// TIA Portal V21 export
// export: Created 2026-07-05T03:49:26.3917626Z, ExportSetting None, DisplayName Totally Integrated Automation Portal, DisplayVersion V21, DisplayName SINAMICS Startdrive Advanced, DisplayVersion V21, DisplayName SINAMICS Startdrive G110M, G120, G120C, G120D, G120P, G115D, DisplayVersion V21, DisplayName SINAMICS Startdrive G130, G150, S120, S150, G200, G220, S200, S210, S220, Innomotics MVD, DisplayVersion V21, DisplayName STEP 7 Professional, DisplayVersion V21, DisplayName STEP 7 Safety, DisplayVersion V21, DisplayName Tech WebApplication, DisplayVersion V21, DisplayName WinCC Basic/Comfort/Advanced, DisplayVersion V21, DisplayName WinCC Professional, DisplayVersion V21, DisplayName WinCC Unified, DisplayVersion V21
FUNCTION_BLOCK "FlowControl_LAD"   // FB2100, LAD
{ S7_Optimized_Access := 'TRUE' }
// stored: AutoNumber false, MemoryReserve 100, SetENOAutomatically false
   VAR_INPUT
      启用 : Bool;   // 使能流程控制FB，FALSE时不允许启动
      启动 : Bool;   // 启动命令，条件满足时进入步骤1
      停止 : Bool;   // 正常停止命令，停止运行并把当前步清零
      暂停 : Bool;   // 暂停命令，保持当前步不继续推进
      复位 : Bool;   // 复位命令，清除完成/故障/暂停并把当前步清零
      中止 : Bool;   // 中止命令，强制退出流程并把当前步清零
      启动允许 : Bool;   // 启动允许条件，例如安全、气压、伺服Ready等
      联锁正常 : Bool;   // 运行中联锁正常，FALSE时触发故障
   END_VAR
   VAR_OUTPUT
      就绪 : Bool;   // 可启动状态：启用、允许、无运行、无故障、未完成
      运行中 : Bool;   // 流程运行锁存状态
      完成 : Bool;   // 流程正常完成，需要复位清除
      故障 : Bool;   // 流程异常停止，需要复位清除
      已暂停 : Bool;   // 流程暂停锁存状态
      当前步 : Int;   // 当前流程步骤号，流程段直接MOVE维护
      故障代码 : Word;   // 故障代码，257表示运行中联锁断开
   END_VAR
   VAR
      启动边沿 : Bool;   // 启动P上升沿指令的边沿存储位
      完成边沿 : Bool;   // 完成P上升沿线圈的边沿存储位
      执行条件 : Bool;   // 运行中和未暂停映射给执行条件
      IEC_Timer_0_Instance { S7_SetPoint := 'True'} : TON_TIME;
      IEC_Timer_0_Instance_1 { S7_SetPoint := 'True'} : TON_TIME;
   END_VAR
   VAR_TEMP   // added for the SCL form of the ladder/FBD networks
      _w1 : Bool;
      _w2 : Bool;
   END_VAR
BEGIN

REGION Network 1: 复位或中止清除流程状态
   // 复位或中止时一次性清除运行、暂停、完成、故障、当前步和故障代码。
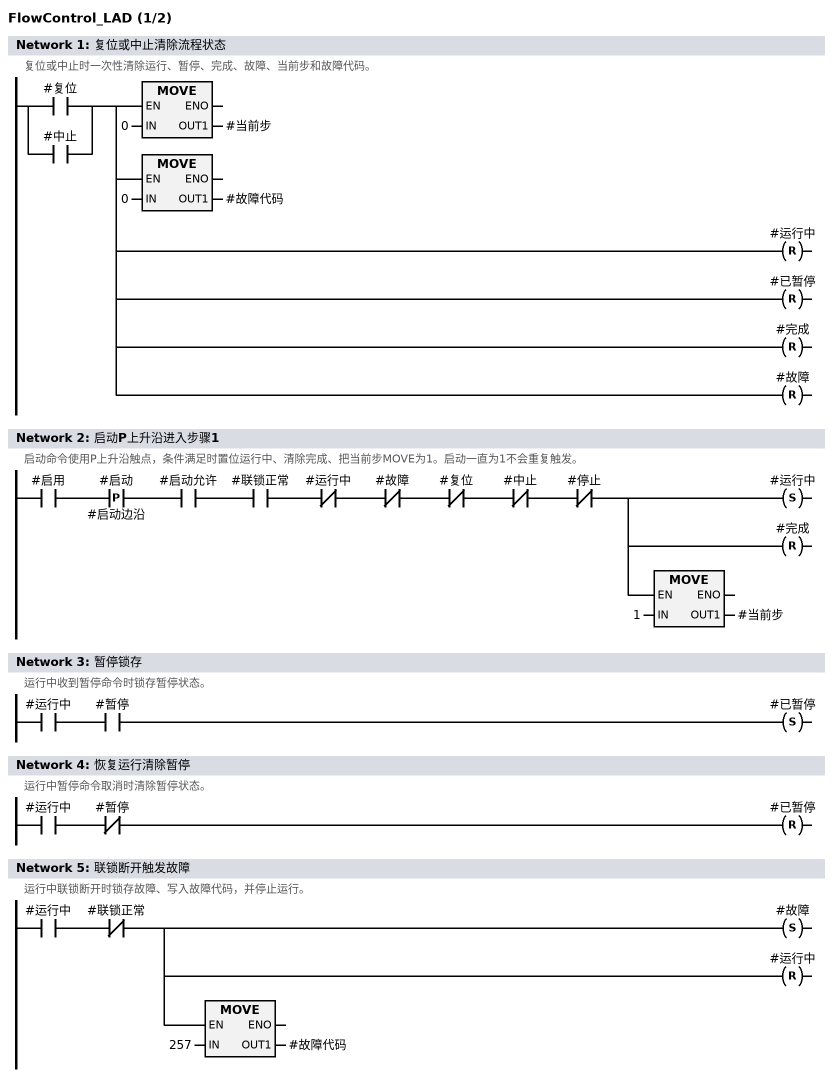
   RUNG wire#powerrail
      Contact( #复位 )
      wire#w1
      { S7_GenerateENO := "TRUE" } Move(in := 0, out1 => #当前步)
   END_RUNG
   RUNG wire#powerrail
      Contact( #中止 )
   END_RUNG wire#w1
   RUNG wire#w1
      { S7_GenerateENO := "TRUE" } Move(in := 0, out1 => #故障代码)
   END_RUNG
   RUNG wire#w1
      R_Coil( #运行中 )
   END_RUNG
   RUNG wire#w1
      R_Coil( #已暂停 )
   END_RUNG
   RUNG wire#w1
      R_Coil( #完成 )
   END_RUNG
   RUNG wire#w1
      R_Coil( #故障 )
   END_RUNG
   // the same network as SCL:
   IF #复位 OR #中止 THEN
       #当前步 := 0;
       #故障代码 := 0;
       #运行中 := FALSE;
       #已暂停 := FALSE;
       #完成 := FALSE;
       #故障 := FALSE;
   END_IF;
END_REGION

REGION Network 2: 启动P上升沿进入步骤1
   // 启动命令使用P上升沿触点，条件满足时置位运行中、清除完成、把当前步MOVE为1。启动一直为1不会重复触发。
   RUNG wire#powerrail
      Contact( #启用 )
      P_Contact(operand := #启动, bit := #启动边沿)
      Contact( #启动允许 )
      Contact( #联锁正常 )
      I_Contact( #运行中 )
      I_Contact( #故障 )
      I_Contact( #复位 )
      I_Contact( #中止 )
      I_Contact( #停止 )
      wire#w1
      S_Coil( #运行中 )
   END_RUNG
   RUNG wire#w1
      R_Coil( #完成 )
   END_RUNG
   RUNG wire#w1
      { S7_GenerateENO := "TRUE" } Move(in := 1, out1 => #当前步)
   END_RUNG
   // the same network as SCL:
   #_w1 := #启用 AND #启动 AND NOT #启动边沿;   // rising edge of #启动
   #启动边沿 := #启动;
   #_w2 := #_w1 AND #启动允许 AND #联锁正常 AND NOT #运行中 AND NOT #故障 AND NOT #复位 AND NOT #中止 AND NOT #停止;
   IF #_w2 THEN
       #运行中 := TRUE;
       #完成 := FALSE;
       #当前步 := 1;
   END_IF;
END_REGION

REGION Network 3: 暂停锁存
   // 运行中收到暂停命令时锁存暂停状态。
   RUNG wire#powerrail
      Contact( #运行中 )
      Contact( #暂停 )
      S_Coil( #已暂停 )
   END_RUNG
   // the same network as SCL:
   IF #运行中 AND #暂停 THEN #已暂停 := TRUE; END_IF;
END_REGION

REGION Network 4: 恢复运行清除暂停
   // 运行中暂停命令取消时清除暂停状态。
   RUNG wire#powerrail
      Contact( #运行中 )
      I_Contact( #暂停 )
      R_Coil( #已暂停 )
   END_RUNG
   // the same network as SCL:
   IF #运行中 AND NOT #暂停 THEN #已暂停 := FALSE; END_IF;
END_REGION

REGION Network 5: 联锁断开触发故障
   // 运行中联锁断开时锁存故障、写入故障代码，并停止运行。
   RUNG wire#powerrail
      Contact( #运行中 )
      I_Contact( #联锁正常 )
      wire#w1
      S_Coil( #故障 )
   END_RUNG
   RUNG wire#w1
      R_Coil( #运行中 )
   END_RUNG
   RUNG wire#w1
      { S7_GenerateENO := "TRUE" } Move(in := 257, out1 => #故障代码)
   END_RUNG
   // the same network as SCL:
   IF #运行中 AND NOT #联锁正常 THEN #故障 := TRUE; END_IF;
   #_w1 := #运行中 AND NOT #联锁正常;
   IF #_w1 THEN
       #运行中 := FALSE;
       #故障代码 := 257;
   END_IF;
END_REGION

REGION Network 6: 停止命令停止流程
   // 停止命令复位运行中，并把当前步MOVE为0。
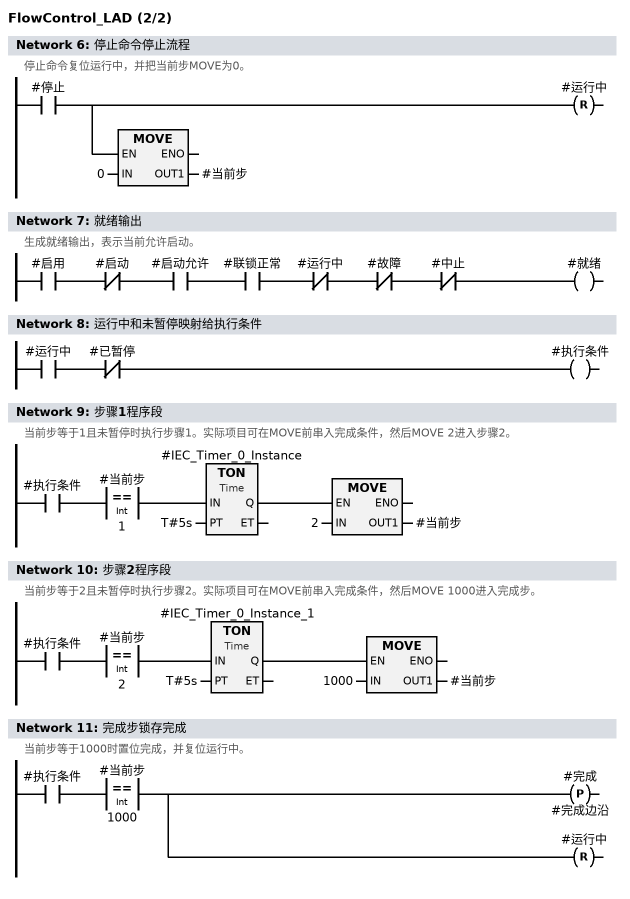
   RUNG wire#powerrail
      Contact( #停止 )
      wire#w1
      R_Coil( #运行中 )
   END_RUNG
   RUNG wire#w1
      { S7_GenerateENO := "TRUE" } Move(in := 0, out1 => #当前步)
   END_RUNG
   // the same network as SCL:
   IF #停止 THEN
       #运行中 := FALSE;
       #当前步 := 0;
   END_IF;
END_REGION

REGION Network 7: 就绪输出
   // 生成就绪输出，表示当前允许启动。
   RUNG wire#powerrail
      Contact( #启用 )
      I_Contact( #启动 )
      Contact( #启动允许 )
      Contact( #联锁正常 )
      I_Contact( #运行中 )
      I_Contact( #故障 )
      I_Contact( #中止 )
      Coil( #就绪 )
   END_RUNG
   // the same network as SCL:
   #就绪 := #启用 AND NOT #启动 AND #启动允许 AND #联锁正常 AND NOT #运行中 AND NOT #故障 AND NOT #中止;
END_REGION

REGION Network 8: 运行中和未暂停映射给执行条件
   RUNG wire#powerrail
      Contact( #运行中 )
      I_Contact( #已暂停 )
      Coil( #执行条件 )
   END_RUNG
   // the same network as SCL:
   #执行条件 := #运行中 AND NOT #已暂停;
END_REGION

REGION Network 9: 步骤1程序段
   // 当前步等于1且未暂停时执行步骤1。实际项目可在MOVE前串入完成条件，然后MOVE 2进入步骤2。
   RUNG wire#powerrail
      Contact( #执行条件 )
      { S7_Templates := "SrcType := Int" } EQ_Contact(in1 := #当前步, in2 := 1)
      { S7_Templates := "time_type := Time" } #IEC_Timer_0_Instance.TON(pt := T#5s, et =>)
      { S7_GenerateENO := "TRUE" } Move(in := 2, out1 => #当前步)
   END_RUNG
   // the same network as SCL:
   #IEC_Timer_0_Instance(IN := #执行条件 AND (#当前步 = 1), PT := T#5s);   // TON
   IF #IEC_Timer_0_Instance.Q THEN #当前步 := 2; END_IF;
END_REGION

REGION Network 10: 步骤2程序段
   // 当前步等于2且未暂停时执行步骤2。实际项目可在MOVE前串入完成条件，然后MOVE 1000进入完成步。
   RUNG wire#powerrail
      Contact( #执行条件 )
      { S7_Templates := "SrcType := Int" } EQ_Contact(in1 := #当前步, in2 := 2)
      { S7_Templates := "time_type := Time" } #IEC_Timer_0_Instance_1.TON(pt := T#5s, et =>)
      { S7_GenerateENO := "TRUE" } Move(in := 1000, out1 => #当前步)
   END_RUNG
   // the same network as SCL:
   #IEC_Timer_0_Instance_1(IN := #执行条件 AND (#当前步 = 2), PT := T#5s);   // TON
   IF #IEC_Timer_0_Instance_1.Q THEN #当前步 := 1000; END_IF;
END_REGION

REGION Network 11: 完成步锁存完成
   // 当前步等于1000时置位完成，并复位运行中。
   #_w1 := #执行条件 AND (#当前步 = 1000);
   #完成 := #_w1 AND NOT #完成边沿;   // rising edge
   #完成边沿 := #_w1;
   IF #_w1 THEN #运行中 := FALSE; END_IF;
END_REGION
END_FUNCTION_BLOCK
